INTERFACE I_Middleware

METHOD Handle
VAR_INPUT
	Request : I_Request;
	Response : I_ServerResponse;
END_VAR
END_METHOD

PROPERTY PUBLIC NextMiddleware : I_Middleware
GET
END_GET
SET
END_SET
END_PROPERTY

END_INTERFACE

(* stored: Version 1.1.0.1, ProductVersion 3.1.4024.12
   Itf I_Middleware: Id {5f09d343-4b6f-4115-a086-1f2a77132465}
   Method Handle: Id {0524a1a2-7537-41f6-b509-fb9c073c5079}
   Property NextMiddleware: Id {667e53a1-2fb3-4f0b-8e53-fe279696cf8f}
   Get Get: Id {ba9318c7-b7ae-47ba-bf09-34529b5a08a0}
   Set Set: Id {e8c500ef-1f06-436e-9258-23c7290e48dd} *)
